// TIA Portal V19 export
DATA_BLOCK "Data"   // DB5
{ S7_Optimized_Access := 'TRUE' }
// stored: MemoryReserve 100
   VAR
      Second : Int;
      Day : Int;
      Mothercores { S7_SetPoint := 'True'} : "array2Months";
      setsProduced { S7_SetPoint := 'True'} : "array2Months";
   END_VAR
BEGIN
END_DATA_BLOCK
